// TIA Portal V17 export
// export: Created 2024-09-02T12:49:54.1271396Z, ExportSetting WithDefaults, DisplayName Totally Integrated Automation Portal, DisplayVersion V17, DisplayName TIA Portal Openness, DisplayVersion V17, DisplayName TIA Portal Version Control Interface, DisplayVersion V17, DisplayName STEP 7 Professional, DisplayVersion V17, DisplayName STEP 7 Safety, DisplayVersion V17, DisplayName WinCC Professional, DisplayVersion V17
DATA_BLOCK "SysDI_Safety"   // DB7001, F_DB
{ DB_Accessible_From_OPC_UA := 'FALSE' }
AUTHOR : FALG1b58
FAMILY : FPRI1b59
NAME : F31b59
VERSION : 0.0
// stored: AutoNumber false, DBAccessibleFromOPCUA false, InstanceOfName AnwFB_Safety, InstanceOfType FB
"AnwFB_Safety"
   // VAR
   //    statTrue : Bool;
   //    statFalse : Bool;
   //    HM_1_ack : Bool;
   //    HM_SK_ack_1 : Bool;
   //    HM_FGroup_ack : Bool;
   //    HM_LC_ack_1 : Bool;
   //    Error_FDback_all { ExternalWritable := 'False'} : Bool;
   //    ACK_Global { S7_SetPoint := 'True'} : ACK_GL;
   //    EStop_1 { S7_SetPoint := 'True'} : ESTOP1;
   //    EStop_2 { S7_SetPoint := 'True'} : ESTOP1;
   //    EStop_3 { S7_SetPoint := 'True'} : ESTOP1;
   //    EStop_4 { S7_SetPoint := 'True'} : ESTOP1;
   //    EStop_5 { S7_SetPoint := 'True'} : ESTOP1;
   //    EStop_6 { S7_SetPoint := 'True'} : ESTOP1;
   //    EStop_7 { S7_SetPoint := 'True'} : ESTOP1;
   //    EStop_8 { S7_SetPoint := 'True'} : ESTOP1;
   //    LC_1 { S7_SetPoint := 'True'} : ESTOP1;
   //    LC_2 { S7_SetPoint := 'True'} : ESTOP1;
   //    LC_3 { S7_SetPoint := 'True'} : ESTOP1;
   //    LC_4 { S7_SetPoint := 'True'} : ESTOP1;
   //    LC_5 { S7_SetPoint := 'True'} : ESTOP1;
   //    LC_MUT_1 { S7_SetPoint := 'True'} : MUT_P;
   //    LC_MUT_2 { S7_SetPoint := 'True'} : MUT_P;
   //    LC_MUT_3 { S7_SetPoint := 'True'} : MUT_P;
   //    LC_MUT_4 { S7_SetPoint := 'True'} : MUT_P;
   //    LC_MUT_5 { S7_SetPoint := 'True'} : MUT_P;
   //    SD_1 { S7_SetPoint := 'True'} : ESTOP1;
   //    SD_2 { S7_SetPoint := 'True'} : ESTOP1;
   //    SD_3 { S7_SetPoint := 'True'} : ESTOP1;
   //    SD_4 { S7_SetPoint := 'True'} : ESTOP1;
   //    SD_5 { S7_SetPoint := 'True'} : ESTOP1;
   //    BR_1 { S7_SetPoint := 'True'} : EV1oo2DI;
   //    BR_2 { S7_SetPoint := 'True'} : EV1oo2DI;
   //    BR_3 { S7_SetPoint := 'True'} : EV1oo2DI;
   //    BR_4 { S7_SetPoint := 'True'} : EV1oo2DI;
   //    BR_5 { S7_SetPoint := 'True'} : EV1oo2DI;
   //    EnblCircuit_01 { S7_SetPoint := 'True'} : FDBACK;
   //    EnblCircuit_02 { S7_SetPoint := 'True'} : FDBACK;
   //    EnblCircuit_03 { S7_SetPoint := 'True'} : FDBACK;
   //    EnblCircuit_04 { S7_SetPoint := 'True'} : FDBACK;
   //    EnblCircuit_05 { S7_SetPoint := 'True'} : FDBACK;
   //    EnblCircuit_06 { S7_SetPoint := 'True'} : FDBACK;
   //    EnblCircuit_07 { S7_SetPoint := 'True'} : FDBACK;
   //    EnblCircuit_08 { S7_SetPoint := 'True'} : FDBACK;
   //    EnblCircuit_09 { S7_SetPoint := 'True'} : FDBACK;
   //    EnblCircuit_10 { S7_SetPoint := 'True'} : FDBACK;
   //    EnblCircuit_11 { S7_SetPoint := 'True'} : FDBACK;
   //    EnblCircuit_12 { S7_SetPoint := 'True'} : FDBACK;
   //    EnblCircuit_13 { S7_SetPoint := 'True'} : FDBACK;
   //    EnblCircuit_14 { S7_SetPoint := 'True'} : FDBACK;
   //    EnblCircuit_15 { S7_SetPoint := 'True'} : FDBACK;
   //    SafetyZone_1 { S7_SetPoint := 'True'} : EV1oo2DI;
   //    SafetyZone_2 { S7_SetPoint := 'True'} : EV1oo2DI;
   //    SafetyZone_3 { S7_SetPoint := 'True'} : EV1oo2DI;
   //    SafetyZone_4 { S7_SetPoint := 'True'} : EV1oo2DI;
   //    SafetyZone_5 { S7_SetPoint := 'True'} : EV1oo2DI;
   //    EnblCircuit_delay_01 { S7_SetPoint := 'True'} : TOF;
   //    EnblCircuit_delay_02 { S7_SetPoint := 'True'} : TOF;
   //    EnblCircuit_delay_03 { S7_SetPoint := 'True'} : TOF;
   //    EnblCircuit_delay_04 { S7_SetPoint := 'True'} : TOF;
   //    EnblCircuit_delay_05 { S7_SetPoint := 'True'} : TOF;
   //    EnblCircuit_delay_06 { S7_SetPoint := 'True'} : TOF;
   //    EnblCircuit_delay_07 { S7_SetPoint := 'True'} : TOF;
   //    EnblCircuit_delay_08 { S7_SetPoint := 'True'} : TOF;
   //    EnblCircuit_delay_09 { S7_SetPoint := 'True'} : TOF;
   //    EnblCircuit_delay_10 { S7_SetPoint := 'True'} : TOF;
   //    EnblCircuit_delay_11 { S7_SetPoint := 'True'} : TOF;
   //    EnblCircuit_delay_12 { S7_SetPoint := 'True'} : TOF;
   //    EnblCircuit_delay_13 { S7_SetPoint := 'True'} : TOF;
   //    EnblCircuit_delay_14 { S7_SetPoint := 'True'} : TOF;
   //    EnblCircuit_delay_15 { S7_SetPoint := 'True'} : TOF;
   // END_VAR
BEGIN
END_DATA_BLOCK
